// TIA Portal V20 export
// export: Created 2026-04-11T06:02:30.785459Z, ExportSetting WithDefaults, DisplayName Totally Integrated Automation Portal, DisplayVersion V20, DisplayName TIA Portal Openness, DisplayVersion V20, DisplayName TIA Portal Version Control Interface, DisplayVersion V20, DisplayName STEP 7 Professional, DisplayVersion V20, DisplayName STEP 7 Safety, DisplayVersion V20, DisplayName WinCC Basic/Comfort/Advanced, DisplayVersion V20, DisplayName WinCC Unified, DisplayVersion V20
TYPE "udtQueueItem"
// stored: IsFailsafeCompliant false
   STRUCT
      bQueueRequest { ExternalWritable := 'False'} : Bool;   // Request to be queued
      iQueuePosition { ExternalWritable := 'False'} : Int;   // Position in the queue
      iPriority { ExternalWritable := 'False'} : Int;   // Priority number, 0 = default/none
   END_STRUCT;
END_TYPE
